//Switchgear
	Monitoringvars.Switchgear.b_NetContactorState 		:= monitor.powerstack.Netcontactor.b_NetConFb;
	Monitoringvars.Switchgear.b_ACInputState 			:= monitor.ACswitchgear.b_InputContactorfb AND monitor.ACswitchgear.b_InputMCCBfb;
	Monitoringvars.Switchgear.b_ACOutputState 			:= monitor.ACswitchgear.b_OutputMCCBfb;
	Monitoringvars.Switchgear.r_ACInputPower 			:= monitor.powermonitor.InputField.ar_Current[0];
	Monitoringvars.Switchgear.r_ACOutputPower 			:= monitor.powermonitor.OutputField.ar_Current[0];
	Monitoringvars.Switchgear.b_ACDetectedBusbar 		:= monitor.powerstack.b_ACDetected;
	Monitoringvars.Switchgear.b_ACDetectedInput 		:= monitor.powermonitor.InputField.e_ACrotationStatus <> 0;
	Monitoringvars.Switchgear.b_DCCouplingState 		:= monitor.DClink.b_DCCouplingState;
	Monitoringvars.Switchgear.b_DCDetected				:= monitor.battery.BatteryInfo.r_SystemVoltage > 120;
	Monitoringvars.Switchgear.r_DCCouplingCurrent 		:= monitor.DClink.Powerdata.Current;
	Monitoringvars.Switchgear.b_PeNeutralLink 			:= monitor.ACswitchgear.b_PENlinkfb;
	Monitoringvars.Switchgear.b_InputSync				:= monitor.ACswitchgear.b_InputSynchronizerfb;
	Monitoringvars.Switchgear.r_ACInputPower			:= monitor.powermonitor.InputField.ar_ActivePower[0];
	Monitoringvars.Switchgear.r_ACOutputPower			:= monitor.powermonitor.OutputField.ar_ActivePower[0];
	Monitoringvars.Switchgear.r_DCCouplingCurrent		:= 0; //monitor.powermonitor.DCbus.?

//Enclosure
	Monitoringvars.enclosure.b_DoorClosedClientPanel 	:= NOT monitor.enclosure.doors.b_ClientpanelDoorOpen;
	Monitoringvars.enclosure.b_DoorClosedControlPanel	:= NOT monitor.enclosure.doors.b_ControlPanelDoorOpen;
	Monitoringvars.enclosure.b_DoorClosedInverter		:= monitor.safety.b_InverterDoorOK;
	Monitoringvars.enclosure.b_HumidityHigh				:= monitor.enclosure.climate.events.b_HumidityHigh;
	Monitoringvars.enclosure.b_HumidityTooHigh			:= monitor.enclosure.climate.events.b_HumidityTooHigh;
	Monitoringvars.enclosure.b_TemperatureHigh			:= monitor.enclosure.climate.events.b_TemperatureHigh;
	Monitoringvars.enclosure.b_TemperatureTooHigh 		:= monitor.enclosure.climate.events.b_TemperatureTooHigh;
	Monitoringvars.enclosure.b_TemperatureLow 			:= monitor.enclosure.climate.events.b_TemperatureLow;
	Monitoringvars.enclosure.b_TemperatureTooLow 		:= monitor.enclosure.climate.events.b_TemperatureTooLow;
	Monitoringvars.enclosure.r_Humidity					:= monitor.enclosure.climate.r_Humidity;
	Monitoringvars.enclosure.r_Temperature 				:= monitor.enclosure.climate.r_Temperature;
	
//Firedetection
	Monitoringvars.firedetection.e_SmokeDetectorState 	:= monitor.protections.FireDetection.SmokeDetectors.State;
	Monitoringvars.firedetection.e_CoDetectorState 		:= monitor.protections.FireDetection.CoDetectors.State;
	Monitoringvars.firedetection.r_CoDetectorLeftValue 	:= monitor.protections.FireDetection.CoDetectors.Value[1];
	Monitoringvars.firedetection.r_CoDetectorRightValue := monitor.protections.FireDetection.CoDetectors.Value[2];
	
//Overcurrent protection
	monitoringvars.OCP.b_InputMCCBstate					:= monitor.ACswitchgear.b_InputMCCBfb;
	monitoringvars.OCP.b_OutputMCCBstate				:= monitor.ACswitchgear.b_OutputMCCBfb;
	monitoringvars.OCP.b_InputOverloadAlarm 			:= monitor.protections.OvercurrentProtection.b_InputAlarm;
	monitoringvars.OCP.b_OutputOverloadAlarm 			:= monitor.protections.OvercurrentProtection.b_OutputAlarm;
	monitoringvars.OCP.b_InputOverloadWarning 			:= monitor.protections.OvercurrentProtection.b_InputWarning;
	monitoringvars.OCP.b_OutputOverloadWarning 			:= monitor.protections.OvercurrentProtection.b_OutputWarning;
	monitoringvars.OCP.r_CurrentPeak 					:= monitor.protections.OvercurrentProtection.r_PeakCurrent;
	monitoringvars.OCP.s_Location 						:= monitor.protections.OvercurrentProtection.s_locationPeak;
	monitoringvars.OCP.t_PeakDuration 					:= monitor.protections.OvercurrentProtection.t_PeakCurrentDuration;
	
//protections
	monitoringvars.protections.b_InsulationOk 			:= monitor.safety.b_InsulationMonitorOK;
	monitoringvars.protections.e_EarthingSystemDetected := monitor.protections.Insulation.e_EarthingSystemDetected;
	monitoringvars.protections.b_InsulationAlarm 		:= NOT monitor.safety.b_InsulationMonitorOK;
	monitoringvars.protections.b_InsulationPenDetected 	:= monitor.protections.Insulation.b_PENlinkDetected;
	monitoringvars.protections.b_InsulationEnable 		:= monitor.protections.Insulation.b_Enabled;
	monitoringvars.protections.b_InsulationWarning 		:= monitor.protections.Insulation.b_Warning;
	monitoringvars.protections.b_MrcdbWarning			:= monitor.protections.MRCDB.b_prewarning;
	monitoringvars.protections.b_MrcdbOK 				:= monitor.safety.b_MRCDBOK;
	monitoringvars.protections.b_MrcdbAlarm 			:= NOT monitor.safety.b_MRCDBOK;
	monitoringvars.protections.b_SurgeType12OK 			:= monitor.protections.Surge.b_Type12_OK;
	monitoringvars.protections.b_SurgeType3OK 			:= monitor.protections.Surge.b_Type3_OK;

	
//UPS
	monitoringvars.UPS.b_BatteryLowCritical				:= monitor.internalpsu.UPS.Events.b_BatteryLowError;
	monitoringvars.UPS.b_BatteryLowWarning				:= monitor.internalpsu.UPS.Events.b_BatteryLowWarning;
	monitoringvars.UPS.b_BatteryLowInfo					:= monitor.internalpsu.UPS.Events.b_BatteryLowInfo;
	monitoringvars.UPS.b_ChargerActive					:= monitor.internalpsu.UPS.b_ChargerActive;
	monitoringvars.UPS.b_InputVoltageFault				:= monitor.internalpsu.UPS.Events.b_InputVoltageWarning;
	monitoringvars.UPS.b_SupplyOnBattery				:= monitor.internalpsu.UPS.b_SystemOnBattery;
	monitoringvars.UPS.r_BatteryVoltage					:= monitor.internalpsu.UPS.r_BatteryVoltage;
	monitoringvars.UPS.r_InputVoltage					:= monitor.internalpsu.UPS.r_InputVoltage;
	monitoringvars.UPS.r_OutputVoltage					:= monitor.internalpsu.UPS.r_OutputVoltage;
	monitoringvars.UPS.r_OutputCurrent					:= monitor.internalpsu.UPS.r_OutputCurrent;
	monitoringvars.UPS.ui_SoC							:= monitor.internalpsu.UPS.ui_SOC;
	
//Internal powersupply
	monitoringvars.IPSU.b_24VdcOK						:= monitor.internalpsu.b_24VdcAvailable;
	monitoringvars.IPSU.b_400VacOK						:= monitor.internalpsu.b_400VACAvailable;
	monitoringvars.IPSU.b_HvdcOK						:= monitor.internalpsu.b_HVDCAvailable;
		
//Zeropoint transformer 
	monitoringvars.ZPT.b_ZPTOverloadAlarm				:= monitor.neutraltransformer.events.b_NeutralCurrentTooHigh;
	monitoringvars.ZPT.b_ZPTOverloadWarning				:= monitor.neutraltransformer.events.b_NeutralCurrentHigh;
	monitoringvars.ZPT.b_VoltageUnbalanceAlarm			:= monitor.neutraltransformer.events.b_VoltageUnbalanceTooHigh;
	monitoringvars.ZPT.b_VoltageUnbalanceWarning		:= monitor.neutraltransformer.events.b_VoltageUnbalanceHigh;
	monitoringvars.ZPT.r_TemperatureL1					:= monitor.neutraltransformer.r_TemperaturePhase[1];
	monitoringvars.ZPT.r_TemperatureL2					:= monitor.neutraltransformer.r_TemperaturePhase[2];
	monitoringvars.ZPT.r_TemperatureL3					:= monitor.neutraltransformer.r_TemperaturePhase[3];
	monitoringvars.ZPT.r_voltageunbalance				:= monitor.powermonitor.OutputField.r_VoltageUnbalance;
	monitoringvars.ZPT.r_powerload						:= monitor.neutraltransformer.r_Powerload;
	monitoringvars.ZPT.b_TempWarningL1					:= monitor.neutraltransformer.events.b_TemperatureHighPhase[1];
	monitoringvars.ZPT.b_TempWarningL2					:= monitor.neutraltransformer.events.b_TemperatureHighPhase[2];
	monitoringvars.ZPT.b_TempWarningL3					:= monitor.neutraltransformer.events.b_TemperatureHighPhase[3];
	monitoringvars.ZPT.b_TempAlarmL1					:= monitor.neutraltransformer.events.b_TemperatureTooHighPhase[1];
	monitoringvars.ZPT.b_TempAlarmL2					:= monitor.neutraltransformer.events.b_TemperatureTooHighPhase[2];
	monitoringvars.ZPT.b_TempAlarmL3					:= monitor.neutraltransformer.events.b_TemperatureTooHighPhase[3];

//connections
	monitoringvars.Connections.b_IoTEnabled				:= Iotcontrolvars.b_Active;
	monitoringvars.Connections.e_IoTConnectionState		:= IoTcontrolvars.e_ConnectionState;
	monitoringvars.Connections.b_ExtControllerEnabled	:= PNcontrolvars.b_Active;
	monitoringvars.Connections.e_ExtConnectionState		:= PNcontrolvars.e_ConnectionState;
	monitoringvars.Connections.s_OutputJson				:= PNcontrolvars.s_OutputJson;
	monitoringvars.Connections.b_PsbOK					:= monitor.peakshavebox.b_buscouplerReady;
	monitoringvars.Connections.e_ActiveController		:= controlvars.HardSettings.setup.e_ControlSource;
	monitoringvars.Connections.e_EthercatState			:= monitor.PLC.e_EthercatState;
	monitoringvars.Connections.e_ProfinetState			:= monitor.PLC.e_ProfinetState;
	monitoringvars.Connections.r_CPUload				:= monitor.PLC.r_CPUload;
	
//battery
	monitoringvars.Battery.r_SoCReal					:= monitor.battery.BatteryInfo.r_SOC;
	monitoringvars.Battery.e_status						:= monitor.battery.BatteryInfo.e_BMS_Status;
	monitoringvars.Battery.r_SocScaled					:= monitor.battery.BatteryInfo.r_SOCScaled;
	monitoringvars.Battery.r_MaxDischargePower			:= monitor.battery.BatteryInfo.r_MaxDischargePowerAllowed;
	monitoringvars.Battery.r_MaxChargePower				:= monitor.battery.BatteryInfo.r_MaxChargePowerAllowed;
	monitoringvars.Battery.r_CellTempMin				:= monitor.battery.BatteryInfo.ar_CellTemperature[eSubValues.Minimum];
	monitoringvars.Battery.r_CellTempMax				:= monitor.battery.BatteryInfo.ar_CellTemperature[eSubValues.Maximum];													
	monitoringvars.Battery.r_CellVoltageMin				:= monitor.battery.BatteryInfo.ar_CellVoltage[eSubValues.Minimum];
	monitoringvars.Battery.r_CellVoltageMax				:= monitor.battery.BatteryInfo.ar_CellVoltage[eSubValues.Maximum];								
	monitoringvars.Battery.r_SoH						:= monitor.battery.BatteryInfo.r_SOH;
	monitoringvars.Battery.r_DCcurrent					:= monitor.battery.BatteryInfo.r_SystemCurrent;
	monitoringvars.Battery.r_DCvoltage					:= monitor.battery.BatteryInfo.r_SystemVoltage;
	monitoringvars.Battery.r_NetRemainingCapacity		:= monitor.battery.BatteryInfo.r_RemainingDischargeEnergyNett;
	monitoringvars.Battery.ui_CycleCount				:= monitor.battery.BatteryInfo.ui_CycleCount;
	
//Powerstack
	monitoringvars.Powerstack.b_ACDetected				:= monitor.powerstack.b_GridACdetected;
	monitoringvars.Powerstack.b_DCDetected				:= monitor.powerstack.b_DCDetected;
	monitoringvars.Powerstack.b_StartedState			:= monitor.powerstack.b_StartedState;
	monitoringvars.Powerstack.b_ControlEnabled			:= monitor.powerstack.b_ControlEnabled;
	monitoringvars.Powerstack.b_MasterEnabled			:= monitor.powerstack.PowermoduleMaster.b_online;
	monitoringvars.Powerstack.b_SlaveEnabled			:= monitor.powerstack.PowermoduleSlave.b_online AND settings.Configuration.b_DoublePowerModule;
	monitoringvars.Powerstack.r_ActivePower				:= monitor.powerstack.r_ActivePower;
	monitoringvars.Powerstack.r_DcPower					:= monitor.powerstack.r_Dcpower;
	monitoringvars.Powerstack.r_Powerload				:= monitor.powerstack.r_LoadPercent;
	monitoringvars.Powerstack.e_MasterState				:= monitor.powerstack.Powermodulemaster.e_Status;
	monitoringvars.Powerstack.e_SlaveState				:= monitor.powerstack.Powermoduleslave.e_Status;
	monitoringvars.Powerstack.b_MasterCurrThrotActive	:= monitor.powerstack.PowermoduleMaster.Events.b_CurrThrottlingActive;
	monitoringvars.Powerstack.b_MasterTempThrotActive	:= monitor.powerstack.PowermoduleMaster.Events.b_TempThrottlingActive;
	monitoringvars.Powerstack.r_MasterthrotValue		:= monitor.powerstack.PowermoduleMaster.r_OverCurrentValue;
	monitoringvars.Powerstack.b_MasterWarning			:= monitor.powerstack.Events.b_MasterWarning;
	monitoringvars.Powerstack.b_MasterMCCBfb			:= monitor.powerstack.PowermoduleMaster.b_MccbFb;
	monitoringvars.Powerstack.b_SlaveCurrThrotActive	:= monitor.powerstack.PowermoduleSlave.Events.b_CurrThrottlingActive;
	monitoringvars.Powerstack.b_SlaveTempThrotActive	:= monitor.powerstack.PowermoduleSlave.Events.b_TempThrottlingActive;
	monitoringvars.Powerstack.r_SlavethrotValue			:= monitor.powerstack.PowermoduleSlave.r_OverCurrentValue;
	monitoringvars.Powerstack.b_SlaveWarning			:= monitor.powerstack.Events.b_SlaveWarning;
	monitoringvars.Powerstack.b_SlaveMCCBfb				:= monitor.powerstack.PowermoduleSlave.b_MccbFb;
	monitoringvars.Powerstack.r_throttlingValue			:= monitor.powerstack.r_OvercurrentValueAct;
	monitoringvars.Powerstack.e_NetContState			:= monitor.powerstack.Netcontactor.e_NetConState;
	monitoringvars.powerstack.e_StatusPowerStack		:= monitor.powerstack.e_State;
	monitoringvars.Powerstack.e_ACrotationState			:= monitor.powermonitor.OutputField.e_ACrotationStatus;
	monitoringvars.Powerstack.b_islandOperation			:= monitor.powerstack.b_InverterGridFormingMode;
	
//Coolingsystem
	monitoringvars.cooling.e_OperationMode 				:= monitor.Cooling.CoolingSystemState;
	monitoringvars.cooling.r_CoolantPressure			:= monitor.Cooling.r_CoolantPressure;
	monitoringvars.cooling.r_CoolantTemperature			:= monitor.Cooling.r_CoolantTemperature;
	monitoringvars.cooling.r_EnclosureDewpoint			:= monitor.Cooling.r_EnclosureDewpoint;
	monitoringvars.cooling.e_HeatPumpStatus				:= monitor.Cooling.HeatPumpStatus;
	monitoringvars.cooling.b_HeatPumpError				:= monitor.Cooling.HeatPumpStatus = eHeatpumpState.ERROR;
	monitoringvars.cooling.b_HeatPumpWarning			:= monitor.Cooling.Events.HeatpumpEvents.b_CommWarning;
	monitoringvars.cooling.b_CoolantPressureError		:= monitor.Cooling.Events.b_CoolingLoopPressureTooLow;
	monitoringvars.cooling.b_CoolantPressureWarning		:= monitor.Cooling.Events.b_CoolingLoopPressureLow;
	monitoringvars.cooling.b_CoolantTempWarning			:= monitor.Cooling.Events.b_CoolantTempLow OR monitor.Cooling.Events.b_CoolantTempHigh;
	
//control feedback
	monitoringvars.controlfb 							:= monitor.controlfb.control;
	
//limits
	monitoringvars.Limits.r_ACcurrentLimit				:= 650;
	monitoringvars.Limits.r_ApparentPowerlimit			:= 450;
	monitoringvars.Limits.r_ActivePowerlimit			:= 360;
	monitoringvars.Limits.r_DCcurrentLimit				:= monitor.battery.BatteryInfo.r_ratedCurrent;
	monitoringvars.limits.r_DroopLimit 					:= settings.MachineParams.Powerstack.r_DroopMaximum;
	
//ConditionalFormatting
	ConditionalFormatting(monitoringvars.ConditionalFormatting, controlvars);
	
//PSB
	monitoringvars.PSB.b_Connected 						:= monitor.peakshavebox.b_buscouplerReady;
	monitoringvars.PSB.b_Active							:= monitor.peakshavebox.b_active;
END_ACTION

METHOD ResetControlvarsOnVariant : BOOL
VAR_INPUT
END_VAR
IF NOT settings.Configuration.b_ACInputConnection THEN
	controlvars.SoftSettings.setup.e_AcInputType := eACInputType.None;
END_IF
END_METHOD

METHOD ResetHMIvarsOnEvent

VAR_INST
	
END_VAR
rTrigResetPowerSetpoints(CLK:= NOT monitor.powerstack.b_StartedState); //monitor.controlfb.HardSettings.setup.e_ControlSource <> 0 OR monitor.system.e_gridmode <> eGridmode.forming);

IF rTrigResetPowerSetpoints.Q THEN
	Controlvars.Operation.system.r_PFset := 1;
	controlvars.Operation.system.r_Pset := 0;
	controlvars.Operation.system.r_Qset := 0;
	controlvars.control.b_start := FALSE;
	controlvars.control.b_stop := FALSE;
END_IF

IF monitor.controlfb.Operation.system.b_GridTakeOverEnable AND monitor.powerstack.b_InverterGridFormingMode THEN
	controlvars.Operation.system.r_Pset := monitor.powerstack.r_ActivePower;
END_IF
END_METHOD

METHOD SetArraydata : BOOL

VAR_IN_OUT
	arrays			: ST_HMI_Monitor_Arraydata;
	init			: BOOL;
END_VAR

VAR_INPUT
	b_sync			: BOOL;
END_VAR

VAR
	index				: INT ;	
END_VAR
IF b_sync OR init THEN
	FOR index := 1 TO (SIZEOF(Arrays.ACInputData) / SIZEOF(st_HMIData)) DO
		DataToHMIArrayFormat(data:= GetAcInputArrayData(data := monitor.powermonitor.inputfield, id:=index), init:= init, st_DataOut := arrays.ACInputData[index]);
	END_FOR
	FOR index := 1 TO (SIZEOF(Arrays.ACOutputData) / SIZEOF(st_HMIData)) DO
		DataToHMIArrayFormat(data:= GetAcOutputArrayData(data := monitor.powermonitor.OutputField, id:=index), init:= init, st_DataOut := arrays.ACOutputData[index]);
	END_FOR
	FOR index := 1 TO (SIZEOF(Arrays.PowerstackData) / SIZEOF(st_HMIData)) DO
		DataToHMIArrayFormat(data:= GetPowerstackArrayData(id:=index), init:= init, st_DataOut := arrays.PowerstackData[index]);
	END_FOR
	FOR index := 1 TO (SIZEOF(Arrays.PmMasterData) / SIZEOF(st_HMIData)) DO
		DataToHMIArrayFormat(data:= GetPowerModuleArrayData(data := monitor.powerstack.PowermoduleMaster, id:=index), init:= init, st_DataOut := arrays.PmMasterData[index]);
	END_FOR
	IF settings.Configuration.b_DcCharger OR INIT THEN
		FOR index := 1 TO (SIZEOF(Arrays.AcDcChargerData) / SIZEOF(st_HMIData)) DO
			DataToHMIArrayFormat(data:= GetDcChargerData(data := monitor.AcDcCharger, id:=index), init:= init, st_DataOut := arrays.AcDcChargerData[index]);
		END_FOR
	END_IF
	IF settings.Configuration.b_DCbuscoupling OR INIT THEN
		FOR index := 1 TO (SIZEOF(Arrays.DcExtension) / SIZEOF(st_HMIData)) DO
			DataToHMIArrayFormat(data:= GetDcExtData(data := monitor.DClink, id:=index), init:= init, st_DataOut := arrays.DcExtension[index]);
		END_FOR
	END_IF
	IF settings.Configuration.b_DoublePowerModule THEN
		FOR index := 1 TO (SIZEOF(Arrays.PmSlaveData) / SIZEOF(st_HMIData)) DO
			DataToHMIArrayFormat(data:= GetPowerModuleArrayData(data := monitor.powerstack.PowermoduleSlave, id:=index), init:= init, st_DataOut := arrays.PmSlaveData[index]);
		END_FOR
	END_IF
	IF settings.MachineParams.GenComm.GenControlProtocol <> 0 OR init THEN
		FOR index := 1 TO (SIZEOF(Arrays.Genset) / SIZEOF(st_HMIData)) DO
			DataToHMIArrayFormat(data:= GetGensetData(data := monitor.Generator, id:=index), init:= init, st_DataOut := arrays.Genset[index]);
		END_FOR
	END_IF
	FOR index := 1 TO (SIZEOF(Arrays.PNcontrolData) / SIZEOF(st_HMIData)) DO
		DataToHMIArrayFormat(data:= GetextcontrolData(data := Pncontrolvars, id:=index), init:= init, st_DataOut := arrays.PNcontrolData[index]);
	END_FOR
	
	FOR index := 1 TO (SIZEOF(Arrays.iotcontrolData) / SIZEOF(st_HMIData)) DO
		DataToHMIArrayFormat(data:= GetextcontrolData(data := IOtcontrolvars, id:=index), init:= init, st_DataOut := arrays.IotcontrolData[index]);
	END_FOR
	FOR index := 1 TO (SIZEOF(Arrays.PSBData) / SIZEOF(st_HMIData)) DO
		DataToHMIArrayFormat(data:= GetPSBData(data := Monitor.peakshavebox, id:=index), init:= init, st_DataOut := arrays.PSBData[index]);
	END_FOR
	FOR index := 1 TO (SIZEOF(Arrays.MBMUdata) / SIZEOF(st_HMIData)) DO
		DataToHMIArrayFormat(data:= GetMBMUData(data := monitor.battery.BatteryInfo, id:=index), init:= init, st_DataOut := arrays.MBMUdata[index]);
	END_FOR
	FOR index := 1 TO (SIZEOF(Arrays.SBMU1data) / SIZEOF(st_HMIData)) DO
		DataToHMIArrayFormat(data:= GetSBMUData(data := monitor.battery.SBMU[0], id:=index, 1), init:= init, st_DataOut := arrays.SBMU1data[index]);
	END_FOR
	FOR index := 1 TO (SIZEOF(Arrays.SBMU2data) / SIZEOF(st_HMIData)) DO
		DataToHMIArrayFormat(data:= GetSBMUData(data := monitor.battery.SBMU[1], id:=index, 2), init:= init, st_DataOut := arrays.SBMU2data[index]);
	END_FOR
	FOR index := 1 TO (SIZEOF(Arrays.SBMU3data) / SIZEOF(st_HMIData)) DO
		DataToHMIArrayFormat(data:= GetSBMUData(data := monitor.battery.SBMU[2], id:=index, 3), init:= init, st_DataOut := arrays.SBMU3data[index]);
	END_FOR
	FOR index := 1 TO (SIZEOF(Arrays.SBMU4data) / SIZEOF(st_HMIData)) DO
		DataToHMIArrayFormat(data:= GetSBMUData(data := monitor.battery.SBMU[3], id:=index, 4), init:= init, st_DataOut := arrays.SBMU4data[index]);
	END_FOR
	FOR index := 1 TO (SIZEOF(Arrays.CoolingSystem) / SIZEOF(st_HMIData)) DO
		DataToHMIArrayFormat(data:= GetCoolingData(data := monitor.Cooling, id:=index), init:= init, st_DataOut := arrays.CoolingSystem[index]);
	END_FOR
// 	FOR index := 1 TO (SIZEOF(Arrays.CoolingSystemHp1) / SIZEOF(st_HMIData)) DO
// 		DataToHMIArrayFormat(data:= GetHeatpumpData(data := monitor.Cooling.HeatPumpSystem.PrimaryHeatpumpGet, id:=index), init:= init, st_DataOut := Arrays.CoolingSystemHp1[index]);
// 	END_FOR
// 	FOR index := 1 TO (SIZEOF(Arrays.CoolingSystemHp2) / SIZEOF(st_HMIData)) DO
// 		DataToHMIArrayFormat(data:= GetHeatpumpData(data := monitor.Cooling.HeatPumpSystem.SecondaryHeatpumpGet, id:=index), init:= init, st_DataOut := Arrays.CoolingSystemHp2[index]);
// 	END_FOR
	
END_IF
END_METHOD

METHOD SettingsChanged : BOOL

VAR_INPUT
	adr1		: DWORD;
	adr2		: DWORD;
	size		: DWORD;
END_VAR

//VAR_IN_OUT CONSTANT
//	hs_user					: ST_hardsettings;
//	hs_PLC					: ST_hardsettings;
	
//END_VAR
SettingsChanged := (MEMCMP(adr1, adr2, size) <> 0);
END_METHOD

END_PROGRAM

(* stored: Version 1.1.0.1, ProductVersion 3.1.4026.18
   POU HMI: Id {60dc6bb9-8218-49aa-8772-c76a0aa4b773}, SpecialFunc None
   Folder ArrayDataMethods: Id {4ca66fc5-9f33-4dca-94c9-22713e87623e}
   Folder ControlsHandlingMethods: Id {9743a59c-d1d0-4ad7-887d-018a332e942f}
   Folder MonitorHandlingMethods: Id {f7a6b299-03d7-4dfc-855c-1ddf6bc9d2c5}
   Folder SchedulerMethods: Id {60f9e2bb-db1c-4499-af8b-7b0818bd2dca}
   Method ConditionalFormatting: Id {d5e65d05-5d3d-4e50-b7f2-4282fc4c1310}
   Method CopyActSettingsFromPLC: Id {326a3b2c-f369-49e3-87db-495557214cc2}
   Method DataToHMIArrayFormat: Id {a405edf0-461d-4789-82bf-da80802179a8}
   Method GetAcInputArrayData: Id {fb71ac2a-7058-4dff-8f7d-bb974837d144}
   Method GetAcOutputArrayData: Id {c030486a-4ccb-4aa0-a2f3-74a767b1f472}
   Method GetActiveTimeSlotScheduler: Id {c40a78b0-a172-4c0a-8e39-5cb8d688ec4d}
   Method GetCoolingData: Id {2d57157c-057a-44c2-b8b2-465df3409131}
   Method GetDcChargerData: Id {351512b6-361a-43ad-b595-ecec3b612c82}
   Method GetDcExtData: Id {d1a8d8de-221f-45ea-a409-c9e3e6332361}
   Method GetextcontrolData: Id {edbeba57-aa21-4dbb-962f-3598133f7234}
   Method GetGensetData: Id {af790907-67b8-4856-92d6-1efbb0af637e}
   Method GetHeatpumpData: Id {ca9d6ad2-f446-421c-b5ea-66fe0797deb9}
   Method GetMBMUData: Id {39578673-79de-4963-a904-8a295803820d}
   Method GetPowerModuleArrayData: Id {58fb203a-814b-4bbe-ad61-b4af9090ca86}
   Method GetPowerstackArrayData: Id {a057df20-bb99-4026-9777-a32c2b8b1466}
   Method GetPSBdata: Id {f976bc01-11eb-4e2f-8e19-f77f419f9bed}
   Method GetSBMUData: Id {355d51c9-ed30-4d57-9a42-70ab2dcd0b09}
   Method Hour_Minute_To_TOW: Id {4fd84871-a229-4c04-9ac1-4641aaa901aa}
   Action MapPLCvarsToHMIVars: Id {1166b49a-6a5d-4f8a-be6d-bc583eb075e4}
   Method ResetControlvarsOnVariant: Id {f7df607d-9743-4bb9-a8dd-30ad9d8c8fd1}
   Method ResetHMIvarsOnEvent: Id {ec0fbc6c-351a-466b-975b-6461819ae91a}
   Method SetArraydata: Id {d229777b-dbdb-4148-ba6c-0979fccd3c91}
   Method SettingsChanged: Id {78c35c0b-34ec-42b9-bcd7-3f10c45fdf5a} *)
